TYPE Axis_STATUS :
STRUCT
	Status : WORD;
	Mode_of_Operation_disp:BYTE;
	Actual_Position:DINT;
	Actual_Velocity :DINT;
	Following_error:DINT;
	Actual_Torque:INT;
END_STRUCT
END_TYPE

(* stored: Version 1.1.0.1, ProductVersion 3.1.4024.12
   DUT Axis_STATUS: Id {bfd2ec8c-2f32-4577-b002-d824088114a6} *)
